FUNCTION_BLOCK FB_Actuation
VAR_INPUT
	bActuation : BOOL;
END_VAR
VAR_OUTPUT
	bDoorUp : BOOL;
	bDoorDown : BOOL;
	
	bDoorLight : BOOL;
END_VAR
VAR
	bDoorOpen : BOOL;
	bDoorClosed : BOOL := TRUE;	// Assumption that in the beginning the door is closed
	bDriveOverload : BOOL;
	
	bPauseWhenOpening : BOOL;
	bPauseWhenClosing : BOOL;
	
	tElapsedClosingTime : TIME;
	tElapsedOpeningTime : TIME;
	
	fbOpeningTimer : TON;
	fbClosingTimer : TON;
	fbLightTimer : TON;
	
	fbActuation : R_TRIG;
	
	fbBlinkingLight : FB_BlinkingLight;

	nCurrentState : DINT;
	
	// Variables needed only for the visualisation
	Rect1 : BOOL;
	Rect2 : BOOL;
	Rect3 : BOOL;
	Rect4 : BOOL;
	Rect5 : BOOL;
	Rect1Time : TIME;
	Rect2Time : TIME;
	Rect3Time : TIME;
	Rect4Time : TIME;
	Rect5Time : TIME;
	bChanged: BOOL;
END_VAR

VAR CONSTANT
	// PT for opening and closing of door timers
	TIMER_PRESET : DWORD := 5000;
	
	// How much time (in ms) should pass in order for the light to turn off when the door has opened / closed 
	LIGHT_DELAY : DWORD := 1000;
	
	// On/off times (in miliseconds) for when the garage door light is blinking in state of error
	BLINKING_TIME_ON : DWORD := 500;
	BLINKING_TIME_OFF : DWORD := 250;
END_VAR

// Rising edge logic in order to stop bouncing (bActuation signal persisting longer than intended)
fbActuation(CLK := bActuation);
bActuation := fbActuation.Q;

CASE nCurrentState OF
	
	0:	// Idle
	
	// If the overload sensor is activated, go to the error state
	IF bDriveOverload THEN
		nCurrentState := 999;
	END_IF
	
	fbOpeningTimer.IN := FALSE;
	fbClosingTimer.IN := FALSE;
	fbLightTimer.IN := FALSE;
	bDoorLight := FALSE;
	
	// If the actuation button is pressed and the door is closed -> open it
	IF bActuation AND (bDoorClosed OR bPauseWhenClosing) THEN
		nCurrentState := 100;
	// If the actuation button is pressed and the door is opened -> close it
	ELSIF bActuation AND (bDoorOpen OR bPauseWhenOpening) THEN
		nCurrentState := 200;
	END_IF
	
	100:	// Opening
	
	// If the overload sensor is activated, say it's paused the opening and go to the error state
	IF bDriveOverload THEN
		bPauseWhenOpening := TRUE;
		bPauseWhenClosing := FALSE;
		tElapsedOpeningTime := fbOpeningTimer.ET;
		nCurrentState := 999;
	END_IF
	
	// Check if the process lasts longer than expected
	IF fbOpeningTimer.ET > TO_TIME(TIMER_PRESET) THEN
		nCurrentState := 999;
	END_IF
	
	// RESET EVERYTHING THAT'S GOTTA DO WITH CLOSING HERE
	bDoorDown := FALSE;
	bDoorClosed := FALSE;
	fbClosingTimer.IN := FALSE;
	
	// State that the door should go up and turn the light on
	bDoorUp := TRUE;
	bDoorLight := TRUE;
	
	// Code needed only for the visualisation
	IF NOT bPauseWhenOpening THEN
		Rect1 := TRUE;
		IF fbOpeningTimer.ET >= Rect2Time THEN
			Rect2 := TRUE;
		END_IF
		IF fbOpeningTimer.ET >= Rect3Time THEN
			Rect3 := TRUE;
		END_IF
		IF fbOpeningTimer.ET >= Rect4Time THEN
			Rect4 := TRUE;
		END_IF
	END_IF
	
	// WRITE TIMER LOGIC FOR OPENING HERE
	fbOpeningTimer.IN := TRUE;
	IF fbOpeningTimer.Q THEN
		bDoorOpen := TRUE;
		bPauseWhenClosing := FALSE;
		
		// Code needed only for the visualisation
		Rect5 := TRUE;
		bChanged := FALSE;
		
		fbLightTimer.IN := TRUE;
		IF fbLightTimer.Q THEN
			bDoorLight := FALSE;
			nCurrentState := 0;
		END_IF		
	END_IF
	
	// The opening is paused -> go to idle state
	IF bActuation THEN
		fbOpeningTimer.IN := FALSE;
		bPauseWhenOpening := TRUE;
		bPauseWhenClosing := FALSE;
		tElapsedOpeningTime := fbOpeningTimer.ET;
	END_IF
	
	IF bPauseWhenOpening THEN
		fbLightTimer.IN := TRUE;
			IF fbLightTimer.Q THEN
				bDoorLight := FALSE;
				nCurrentState := 0;
			END_IF
	END_IF
	
	200:	// Closing
	
	// If the overload sensor is activated, say it's paused the opening and go to the error state
	IF bDriveOverload THEN
		bPauseWhenClosing := TRUE;
		bPauseWhenOpening := FALSE;
		tElapsedClosingTime := fbClosingTimer.ET;
		nCurrentState := 999;
	END_IF
	
	// Check if the process lasts longer than expected
	IF fbClosingTimer.ET > TO_TIME(TIMER_PRESET) THEN
		nCurrentState := 999;
	END_IF
	
	// RESET EVERYTHING THAT'S GOTTA DO WITH OPENING HERE
	bDoorUp := FALSE;
	bDoorOpen := FALSE;
	fbOpeningTimer.IN := FALSE;
	
	// State that the door should go down and turn the light on
	bDoorDown := TRUE;
	bDoorLight := TRUE;
	
	// Code needed only for the visualisation
	IF NOT bPauseWhenClosing THEN
		Rect5 := FALSE;
		IF fbClosingTimer.ET >= Rect2Time THEN
			Rect4 := FALSE;
		END_IF
		IF fbClosingTimer.ET >= Rect3Time THEN
			Rect3 := FALSE;
		END_IF
		IF fbClosingTimer.ET >= Rect4Time THEN
			Rect2 := FALSE;
		END_IF
	END_IF
	
	// WRITE TIMER LOGIC FOR CLOSING HERE
	fbClosingTimer.IN := TRUE;
	IF fbClosingTimer.Q THEN
		bDoorClosed := TRUE;
		bPauseWhenOpening := FALSE;
		
		// Code needed only for the visualisation
		Rect1 := FALSE;
		bChanged := FALSE;
		
		fbLightTimer.IN := TRUE;
		IF fbLightTimer.Q THEN
			bDoorLight := FALSE;
			nCurrentState := 0;
		END_IF
	END_IF
	
	// The closing is paused -> go to idle state
	IF bActuation THEN
		fbClosingTimer.IN := FALSE;
		bPauseWhenClosing := TRUE;
		bPauseWhenOpening := FALSE;
		tElapsedClosingTime := fbClosingTimer.ET;
	END_IF
	
	IF bPauseWhenClosing THEN
		fbLightTimer.IN := TRUE;
			IF fbLightTimer.Q THEN
				bDoorLight := FALSE;
				nCurrentState := 0;
			END_IF
	END_IF
	
	999:	// Error
	
	IF bActuation THEN
		nCurrentState := 0;
	END_IF
	
	fbBlinkingLight(dwTimeOn :=  BLINKING_TIME_ON, dwTimeOff := BLINKING_TIME_OFF, bLight => bDoorLight);
	
	// WRITE LOGIC TO STOP THE WHOLE PROCESS HERE (RESET EVERYTHING)
	bDoorUp := FALSE;
	bDoorDown := FALSE;
	
END_CASE

// Timer presets logic
IF bPauseWhenClosing THEN
	fbOpeningTimer(PT := tElapsedClosingTime);
	
	// Code only needed for the visualisation
	IF NOT bChanged THEN
		IF Rect3 THEN
			Rect4Time := TO_TIME(TO_REAL(tElapsedClosingTime) * 0.5);
			bChanged := TRUE;
		ELSIF Rect2 THEN
			Rect3Time := TO_TIME(TO_REAL(tElapsedClosingTime) * 0.3);
			Rect4Time := TO_TIME(TO_REAL(tElapsedClosingTime) * 0.6);
			bChanged := TRUE;
		ELSIF Rect1 THEN
			Rect2Time := TO_TIME(TO_REAL(tElapsedClosingTime) * 0.25);
			Rect3Time := TO_TIME(TO_REAL(tElapsedClosingTime) * 0.5);
			Rect4Time := TO_TIME(TO_REAL(tElapsedClosingTime) * 0.75);
			bChanged := TRUE;
		END_IF
	END_IF
	
ELSIF bPauseWhenOpening THEN
	fbClosingTimer(PT := tElapsedOpeningTime);
	
	// Code only needed for the visualisation
	IF NOT bChanged THEN
		IF Rect2 THEN
			Rect2Time := TO_TIME(TO_REAL(tElapsedOpeningTime) * 0.25);
			Rect3Time := TO_TIME(TO_REAL(tElapsedOpeningTime) * 0.5);
			Rect4Time := TO_TIME(TO_REAL(tElapsedOpeningTime) * 0.75);
		ELSIF Rect3 THEN
			Rect3Time := TO_TIME(TO_REAL(tElapsedOpeningTime) * 0.3);
			Rect4Time := TO_TIME(TO_REAL(tElapsedOpeningTime) * 0.6);
		ELSIF Rect4 THEN
			Rect4Time := TO_TIME(TO_REAL(tElapsedOpeningTime) * 0.5);
		END_IF
	END_IF

ELSE
	fbOpeningTimer(PT := TO_TIME(TIMER_PRESET));
	fbClosingTimer(PT := TO_TIME(TIMER_PRESET));
	
	// Code only needed for the visualisation
	Rect1Time := TO_TIME(TIMER_PRESET) * 0;
	Rect2Time := TO_TIME(TO_REAL(TIMER_PRESET) * 0.25);
	Rect3Time := TO_TIME(TO_REAL(TIMER_PRESET) * 0.5);
	Rect4Time := TO_TIME(TO_REAL(TIMER_PRESET) * 0.75);
	Rect5Time := TO_TIME(TIMER_PRESET) * 1;
END_IF

fbLightTimer(PT := TO_TIME(LIGHT_DELAY));

END_FUNCTION_BLOCK

(* stored: Version 1.1.0.1, ProductVersion 3.1.4024.12
   POU FB_Actuation: Id {0bcd839f-995b-44ae-a7ea-68a300cc7b56}, SpecialFunc None *)
